// LS Electric XG5000 project: 터치
// PLC LSPLC

PROGRAM NewProgram (task: 스캔 프로그램)

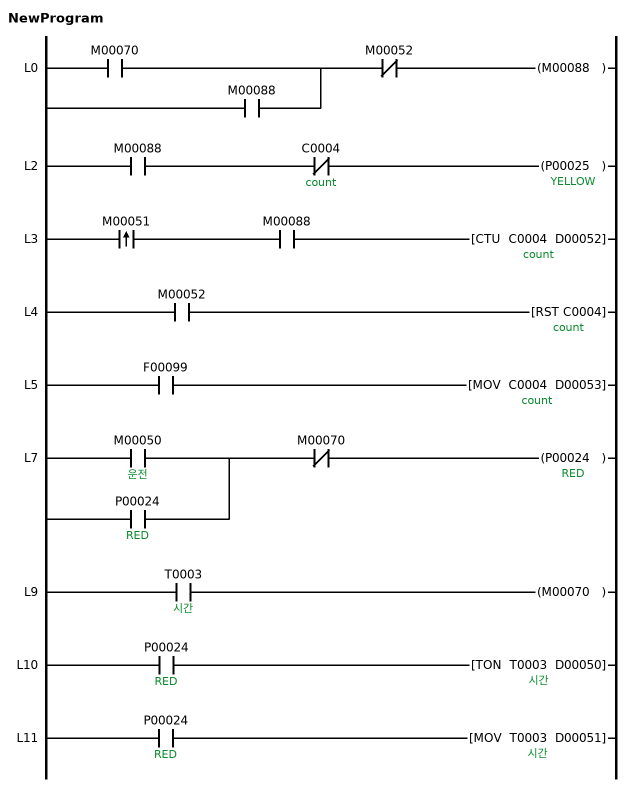
; L0
LOAD      M00070
OR        M00088
AND NOT   M00052
OUT       M00088
; L2
LOAD      M00088
AND NOT   C0004	// count
OUT       P00025	// YELLOW
; L3
LOADP     M00051
AND       M00088
CTU       C0004 D00052	// count
; L4
LOAD      M00052
RST       C0004	// count
; L5
LOAD      F00099
MOV       C0004 D00053	// count
; L7
LOAD      M00050	// 운전
OR        P00024	// RED
AND NOT   M00070
OUT       P00024	// RED
; L9
LOAD      T0003	// 시간
OUT       M00070
; L10
LOAD      P00024	// RED
TON       T0003 D00050	// 시간
; L11
LOAD      P00024	// RED
MOV       T0003 D00051	// 시간

VARIABLES AND COMMENTS (devices not used above)
M00000	BIT	수동/자동
P00020	BIT	전진1
M00011	BIT	1.수동후진
M00101	BIT	1.수동후진
M00100	BIT	1.수동전진
M00010	BIT	1.수동전진
M00012	BIT	2.수동전진
M00102	BIT	2.수동전진
M00013	BIT	2.수동후진
M00103	BIT	2.수동후진
P00022	BIT	전진2
P00021	BIT	후진1
P00023	BIT	후진2
M00002	BIT	자동운전
P00002	BIT	2.후진감지
P00000	BIT	1.후진감지
M00200	BIT	1.전진
P00001	BIT	1.전진감지
M00201	BIT	2.전진
M00202	BIT	1.후진
P00003	BIT	2.전진감지
M00203	BIT	2.후진
M00204	BIT	2.후진완료
M00001	BIT	단속/연속
M00003	BIT	정지
M00004	BIT	리셋
M00005	BIT	일시정지
M00006	BIT	Ready
M00007	BIT	운전중
M00205	BIT	1.후진완료
M00020	BIT	운전
T0000	BIT/WORD	T_ON
P00026	BIT	Toff
T0001	BIT/WORD	Toff
D00000	WORD	d0
M00041	BIT	next
M00042	BIT	Reset